(* IEC 61131-3 sources: ST_DesignPattern/Creational, 7 files *)

(* ---- abstract_factory_pattern.st ---- *)
{attribute 'qualified_only'}
{attribute 'strict'}
TYPE E_Color:
(
	init := 0,
	Black ,
	Red,
	Yellow,
	end
);
END_TYPE

{attribute 'qualified_only'}
{attribute 'strict'}
TYPE E_Shape:
(
	init := 0,
	Circle,
	Rectangle,
	Sqaure,
	Star,
	Triangle,
	end,
	Custom
);
END_TYPE

{attribute 'qualified_only'}
{attribute 'strict'}
TYPE E_Factory:
(
	init := 0,
	Shape,
	Color,
	end
);
END_TYPE

INTERFACE I_Color
    METHOD M_Fill: BOOL
    END_METHOD
END_INTERFACE

INTERFACE I_Shape
    METHOD M_Draw: BOOL
    END_METHOD
END_INTERFACE

FUNCTION_BLOCK FB_Black IMPLEMENTS I_Color
    METHOD M_Fill: BOOL
        ADSLOGSTR(ADSLOG_MSGTYPE_HINT, 'Paint Black', '');
        M_Fill := TRUE;
    END_METHOD
END_FUNCTION_BLOCK

FUNCTION_BLOCK FB_Red IMPLEMENTS I_Color
    METHOD M_Fill: BOOL
        ADSLOGSTR(ADSLOG_MSGTYPE_HINT, 'Paint Red', '');
        M_Fill := TRUE;
    END_METHOD
END_FUNCTION_BLOCK

FUNCTION_BLOCK FB_Yellow IMPLEMENTS I_Color
    METHOD M_Fill: BOOL
        ADSLOGSTR(ADSLOG_MSGTYPE_HINT, 'Paint Yellow', '');
        M_Fill := TRUE;
    END_METHOD
END_FUNCTION_BLOCK

FUNCTION_BLOCK FB_Circle IMPLEMENTS I_Shape
    METHOD M_Draw: BOOL
        ADSLOGSTR(ADSLOG_MSGTYPE_HINT, 'Draw circle', '');
        M_Draw := TRUE;
    END_METHOD
END_FUNCTION_BLOCK

FUNCTION_BLOCK FB_Rectangle IMPLEMENTS I_Shape
    METHOD M_Draw: BOOL
            ADSLOGSTR(ADSLOG_MSGTYPE_HINT, 'Draw rectangle', '');
            M_Draw := TRUE;
    END_METHOD
END_FUNCTION_BLOCK

FUNCTION_BLOCK FB_Sqaure IMPLEMENTS I_Shape
    METHOD M_Draw: BOOL
        ADSLOGSTR(ADSLOG_MSGTYPE_HINT, 'Draw square', '');
        M_Draw := TRUE;
    END_METHOD
END_FUNCTION_BLOCK

FUNCTION_BLOCK FB_Star IMPLEMENTS I_Shape
    METHOD M_Draw: BOOL
        ADSLOGSTR(ADSLOG_MSGTYPE_HINT, 'Draw star', '');
        M_Draw := TRUE;
    END_METHOD
END_FUNCTION_BLOCK

FUNCTION_BLOCK FB_Triangle IMPLEMENTS I_Shape
    METHOD M_Draw: BOOL
        ADSLOGSTR(ADSLOG_MSGTYPE_HINT, 'Draw triangle', '');
        M_Draw := TRUE;
    END_METHOD
END_FUNCTION_BLOCK

FUNCTION_BLOCK ABSTRACT FB_AbstractFactory
    METHOD M_GetColorObject: I_Color
    VAR_INPUT
        eColor: E_Color;
    END_VAR
    END_METHOD

    METHOD M_GetShapeObject: I_Shape
    VAR_INPUT
        eShape: E_Shape;
    END_VAR
    END_METHOD

    METHOD ABSTRACT M_ReleaseMemory: BOOL
    END_METHOD
END_FUNCTION_BLOCK

{attribute 'hide_all_locals'}
{attribute 'enable_dynamic_creation'}
FUNCTION_BLOCK FB_ColorCreator EXTENDS FB_AbstractFactory
    VAR
        pBlack: POINTER TO FB_Black;
        pRed: POINTER TO FB_Red;
        pCircle: POINTER TO FB_Circle;
        iColor: I_Color;
    END_VAR
    METHOD M_GetColorObject: I_Color
    VAR_INPUT
        eColor: E_Color;
    END_VAR
        CASE eColor OF:
            Black:

                // Dynamic instantiation
                pBlack := __NEW(FB_Black);
                iColor := pBlack^;

                // Return the object
                IF iColor <> 0 THEN
                    M_GetColorObject := iColor;
                END_IF

                eColor := E_Color.init;

            Red:

                // Dynamic instantiation
                pRed := __NEW(FB_Red);
                iColor := pRed^;

                // Return the object
                IF iColor <> 0 THEN
                    M_GetColorObject := iColor;
                END_IF

                eColor := E_Color.init;

            Yellow:

                // Dynamic instantiation
                pYellow := __NEW(FB_Yellow);
                iColor := pYellow^;

                // Return the object
                IF iColor <> 0 THEN
                    M_GetColorObject := iColor;
                END_IF

                eColor := E_Color.init;
        END_CASE
    END_METHOD

    METHOD M_ReleaseMemory
        // Release the memory
        IF (pBlack <> 0) THEN
            __DELETE(pBlack);
            pBlack := 0;
        END_IF

        // Release the memory
        IF (pRed <> 0) THEN
            __DELETE(pRed);
            pRed := 0;
        END_IF

        // Release the memory
        IF (pYellow <> 0) THEN
            __DELETE(pYellow);
            pYellow := 0;
        END_IF
    END_METHOD

    METHOD FB_exit
        M_ReleaseMemory();
    END_METHOD
END_FUNCTION_BLOCK

{attribute 'hide_all_locals'}
{attribute 'enable_dynamic_creation'}
FUNCTION_BLOCK FB_ShapeCreator EXTENDS FB_AbstractFactory
VAR
      pCircle: POINTER TO FB_Circle;
      pRectangle: POINTER TO FB_Rectangle;
      pSquare: POINTER TO FB_Square;
      pStar: POINTER TO FB_Star;
      pTriangle: POINTER TO FB_Triangle;
      iShape: I_Shape;
END_VAR

    METHOD M_GetShapeObject: I_shape
    VAR_INPUT
        eShape: E_Shape;
    END_VAR
        CASE eShape OF
            E_Shape.Circle:

                // Dynamic instantiation
                pCircle := __NEW(FB_Circle);
                iShape := pCircle^;

                // Return the object
                IF iShape <> 0 THEN
                    M_GetShapeObject := iShape;
                END_IF

                // Release the memory
                IF (pCircle <> 0) THEN
                    __DELETE(pCircle);
                    pCircle := 0;
                END_IF

                eShape := E_Shape.init;

            E_Shape.Rectangle:
                pRectangle := __NEW(FB_Rectangle);
                iShape := pRectangle^;

                // Return the object
                IF iShape <> 0 THEN
                    M_GetShapeObject := iShape;
                END_IF

                IF (pRectangle <> 0) THEN
                    __DELETE(pRectangle);
                    pRectangle := 0;
                END_IF

                eShape := E_Shape.init;

            E_Shape.Sqaure:
                pSquare := __NEW(FB_Square);
                iShape := pSquare^;

                // Return the object
                IF iShape <> 0 THEN
                    M_GetShapeObject := iShape;
                END_IF

                IF (pSquare <> 0) THEN
                    __DELETE(pSquare);
                    pSquare := 0;
                END_IF

                eShape := E_Shape.init;

            E_Shape.Star:
                pStar := __NEW(FB_Star);
                iShape := pStar^;

                // Return the object
                IF iShape <> 0 THEN
                    M_GetShapeObject := iShape;
                END_IF

                IF (pStar <> 0) THEN
                    __DELETE(pStar);
                    pStar := 0;
                END_IF

                eShape := E_Shape.init;

            E_Shape.Triangle:
                pTriangle := __NEW(FB_Triangle);
                iShape := pTriangle^;

                // Return the object
                IF iShape <> 0 THEN
                    M_GetShapeObject := iShape;
                END_IF

                IF (pTriangle <> 0) THEN
                    __DELETE(pTriangle);
                    pTriangle := 0;
                END_IF

                eShape := E_Shape.init;
        END_CASE
    END_METHOD

    METHOD M_ReleaseMemory: BOOL
    VAR_INPUT
    END_VAR
        IF (pCircle <> 0) THEN
            __DELETE(pCircle);
            pCircle := 0;
        END_IF

        IF (pRectangle <> 0) THEN
            __DELETE(pRectangle);
            pRectangle := 0;
        END_IF

        IF (pSquare <> 0) THEN
            __DELETE(pSquare);
            pSquare := 0;
        END_IF

        IF (pStar <> 0) THEN
            __DELETE(pStar);
            pStar := 0;
        END_IF

        IF (pTriangle <> 0) THEN
            __DELETE(pTriangle);
            pTriangle := 0;
        END_IF
    END_METHOD

    METHOD FB_exit: BOOL
    VAR_INPUT
        bInCopyCode: BOOL; // if TRUE, the exit method is called for exiting an instance that is copied afterwards (online change).
    END_VAR
        M_ReleaseMemory();
    END_METHOD
END_FUNCTION_BLOCK

FUNCTION_BLOCK FB_ShapeCreatorEX EXTENDS FB_ShapeCreator
VAR
	pCustomShape: POINTER TO FB_CustomShape;
END_VAR
    METHOD M_GetShapeObject: I_shape
        IF eShape = E_Shape.Custom THEN

            // Dynamic instantiation
            pCustomShape := __NEW(FB_CustomShape);
            iShape := pCustomShape^;

            // Return the object
            IF iShape <> 0 THEN
                M_GetShapeObject := iShape;
            END_IF

            // Release the memory
            IF (pCustomShape <> 0) THEN
                __DELETE(pCustomShape);
                pCustomShape := 0;
            END_IF

            eShape := E_Shape.init;
        ELSE
            M_GetShapeObject := SUPER^.M_GetShapeObject(eShape);
        END_IF
    END_METHOD
END_FUNCTION_BLOCK

FUNCTION_BLOCK FB_FactoryProducer
VAR
    pColorFactory: POINTER TO FB_ColorCreator;
    pShapeFactory: POINTER TO FB_ShapeCreator;
END_VAR
    METHOD M_GetFactory: REFERENCE TO FB_AbstractFactory
    VAR_INPUT
        eFactory: E_Factory;
    END_VAR
        CASE eFactory OF
            E_Factory.Color:

                pColorFactory := __NEW(FB_ColorCreator);
                IF pColorFactory <> 0 THEN
                    M_GetFactory REF= (pColorFactoy^);
                END_IF

                eFactory := E_Factory.init;

            E_Factory.Shape:

                pShapeFactory := __NEW(FB_ShapeCreator);
                IF pShapeFactory <> 0 THEN
                    M_GetFactory REF = (pShapeFactory^);
                END_IF

                eFactory := E_Factory.init;
        END_CASE
    END_METHOD

    METHOD M_ReleaseMemory: BOOL
        IF pColorFactoy <> 0 THEN
            __DELETE(pColorFactoy);
            pColorFactoy := 0;
        END_IF

        IF pShapeFactory <> 0 THEN
            __DELETE(pShapeFactory);
            pShapeFactory := 0;
        END_IF
    END_METHOD

    METHOD FB_exit: BOOL
    VAR_INPUT
        bInCopyCode: BOOL; // if TRUE, the exit method is called for exiting an instance that is copied afterwards (online change).
    END_VAR
        M_ReleaseMemory();
    END_METHOD
END_FUNCTION_BLOCK

PROGRAM MAIN
VAR
    fbFactoryProducer: FB_FactoryProducer;
    fbFactory: REFERENCE TO FB_AbstractFactory;

    iShape: I_Shape;
    iColor: I_Color;

    eShape: E_Shape := E_Shape.Star;
    eColor: E_Color := E_Color.Red;

    bStart1: BOOL;
    bStart2: BOOL;
END_VAR

IF bStart1 THEN
    // Draw
    fbFactory REF = fbFactoryProducer.M_GetFactory(eFactory := E_Factory.Shape);

    IF __ISVALIDREF(fbFactory) THEN
        iShape := fbFactory.M_GetShapeObject(eShape := eShape);
    END_IF

    IF iShape <> 0 THEN
		iShape.M_Draw();
	END_IF

    // Fill
    fbFactory REF = fbFactoryProducer.M_GetFactory(eFactory := E_Factory.Color);

    IF __ISVALIDREF(fbFactory) THEN
        iColor := fbFactory.M_GetColorObject(eColor := eColor);
    END_IF

    IF iColor <> 0 THEN
		iColor.M_Fill();
	END_IF

    // Release Memory
    fbFactoryProducer.M_ReleaseMemory();

    bStart1 := FALSE;
END_IF
// Alternatively, you can chain the methods and get the same result:
IF bStart2 THEN
	fbFactoryProducer.M_GetFactory(eFactory := E_Factory.Shape).M_GetShapeObject(eShape := eShape).M_Draw();
	fbFactoryProducer.M_GetFactory(eFactory := E_Factory.Color).M_GetColorObject(eColor := eColor).M_Fill();

	// Release Memory
	fbFactoryProducer.M_ReleaseMemory();
	bStart2 := FALSE;
END_IF
END_PROGRAM

(* ---- builder_patter_example1.st ---- *)
///The class Product is just a plain bluprint of the components of the object to be built.
///The final Product may ot may not contain the all the Parts listed on the Product declaration
/// rather only the parts in the specifications sent by the client.
{attribute 'enable_dynamic_creation' := ''}
FUNCTION_BLOCK Product
VAR_INPUT
	///List of possible parts to be build in a final Product object
	mainPart: STRING;
	part1: STRING;
	part2: STRING;
	part3: STRING;
END_VAR
    ///Method to be used in the visualization element for an easier String handling
    METHOD toString : STRING
    VAR
        ///Local variable to join together and store the pieces of String
        tempString: STRING;
    END_VAR
        //tempString joins together "Main Part" and "Part 1" of the Product object
        tempString := CONCAT(THIS^.mainPart , THIS^.part1);
        //tempString joins together its current value and "Part 2" of the Product object
        tempString := CONCAT(tempString , THIS^.part2);
        //tempString joins together its current value and "Part 3" of the Product object
        tempString := CONCAT(tempString , THIS^.part3);
        //The final result is sent as the output of this method
        toString := tempString;
    END_METHOD
END_FUNCTION_BLOCK

///Builder interface to declare all needed parts to be built
INTERFACE ITF_Builder
    ///Illustrative method of the pattern to set the main part
    METHOD Set_Main_Part
    VAR_INPUT
        ///Illustrative value (object because it is a TRING) to be set as a product part
        mainPart: STRING;
    END_VAR

    ///Illustrative method of the pattern to set the part1
    METHOD Set_Part1
    VAR_INPUT
        ///Illustrative value (object because it is a TRING) to be set as a product part
        part1: STRING;
    END_VAR

    ///Illustrative method of the pattern to set the part2
    METHOD Set_Part2
    VAR_INPUT
        ///Illustrative value (object because it is a TRING) to be set as a product part
        part2: STRING;
    END_VAR

    ///Illustrative method of the pattern to set the part3
    METHOD Set_Part3
    VAR_INPUT
        ///Illustrative value (object because it is a TRING) to be set as a product part
        part3: STRING;
    END_VAR
END_INTERFACE

///This is the concrete builder class, reponsible for building the final product object
FUNCTION_BLOCK ConcreteBuilder IMPLEMENTS ITF_Builder
VAR
	///Holds an internal reference to how the final product shoud be so the builder class can build it on the fly /// Contiene una referencia interna sobre cómo debe ser el producto final para que la clase constructora pueda construirlo sobre la marcha.
	/// without any help from other classes exepting the Director class that is going to be passing the special /// sin ninguna ayuda de otras clases excepto la clase Director que va a pasar el especial
	///specifications to the builder.///especificaciones para el constructor.
	localProduct: Product;
	///Stores the specifications, sent by the client, of the final product to be built.
	///Almacena las especificaciones, enviadas por el cliente, del producto final a construir.
	specifications: ARRAY[1..4] OF STRING;
END_VAR

METHOD fb_init
VAR_INPUT
	/// TRUE: the Retain-variables are initialized (reset warm / reset cold)
	bInitRetains: BOOL;
	/// TRUE  the instance will be copied to the copy-code afterward (online change)
	bInCopyCode: BOOL;
	///The constructor receives the specifications for this ConcreteBuilder instance
	///Just in case the concrete builder could change the specifications in the future, otherwise
	/// this specifications should be constant.
	specs: ARRAY[1..4] OF STRING;
END_VAR

    //Stores the specifications on its own specifications field.
    THIS^.specifications := specs;

END_METHOD

///Illustrative method of the pattern to get the main part
METHOD Get_Main_Part : STRING
    //Returns the object stored in the built product THIS^.localProduct.mainPart
    Get_Main_Part := THIS^.localProduct.mainPart;
END_METHOD

///Illustrative method of the pattern
METHOD Get_Result : Product
    //The concrete builder, after it builts the final object of class product, returns the
    // final product object
    Get_Result := THIS^.localProduct;
END_METHOD

///Illustrative method of the pattern to set the part1
METHOD Set_Part1
VAR_INPUT
	///Illustrative value (object because it is a TRING) to be set as a product part
	part1: STRING;
END_VAR
    //Sets the passed value to its corresponding field.
    //We can say that the the final product is in process of being built.
    //So this is a step into building the final product done by the builder.
    THIS^.localProduct.part1 := part1;
END_METHOD

END_FUNCTION_BLOCK

///The director class is responsible to delegate the construction of the final product object
/// to a concrete builder object.
{attribute 'enable_dynamic_creation' := ''}
FUNCTION_BLOCK Director
VAR_INPUT
	///Reference to the builder that is going to be building the final product object.
	///Referencia al constructor que construirá el objeto del producto final.
	{attribute 'old_input_assignments' := ''}
	inputConcreteBuilder: ConcreteBuilder(specs := inputConcreteBuilder.specifications);
END_VAR
VAR
	///Holds a reference to the concrete builder object to send the specifications of the final product to it.
	/// Contiene una referencia al objeto constructor concreto para enviarle las especificaciones del producto final
	{attribute 'old_input_assignments' := ''}
	concreteBuilder: ConcreteBuilder(specs := THIS^.concreteBuilder.specifications);
END_VAR
    //Stores the reference to which builder will be building the final product object in its own field THIS^.concreteBuilder
    //Almacena la referencia a qué constructor construirá el objeto del producto final en su propio campo THIS^.concreteBuilder
    THIS^.concreteBuilder := inputConcreteBuilder;

///This constructor is called at instanciation it is necessary to instanciate the Director instance.
///The specifications of the concreteBuilder instance stored in the Director instance should be set first by the client
/// otherwise a Data Recursion error is caused
METHOD fb_init
VAR_INPUT
	/// TRUE: the Retain-variables are initialized (reset warm / reset cold)
	bInitRetains: BOOL;
	/// TRUE  the instance will be copied to the copy-code afterward (online change)
	bInCopyCode: BOOL;
	///Reference a concreteBuilder instance to instanciate the Director.
	{attribute 'old_input_assignments' := ''}
	inputConcreteBuilder: ConcreteBuilder(specs := defaultArray);
END_VAR
VAR
	///Variable to isntanciate the concreteBuilder instance on the input section. It does not affect the Directors instanciation.
	defaultArray: ARRAY[1..4] OF STRING := ['Default', 'Default', 'Default', 'Default'];
END_VAR
    //Creates the concreteBuilder instance that will be building the final product object in its own field THIS^.concreteBuilder
    //This instance is empty because we can not use Data Recursion with the inputConcreteInstance instanciation.
    //So this concreteBuilder instance should be changed by the client before a Construct() request is called on the Director for the first time only.
    THIS^.concreteBuilder := inputConcreteBuilder;
END_METHOD

///This method is going to be called by the client when a new Product object must be built
METHOD Construct : Product
    //The Director tells its concreteBuilder instance to build the final product step by step passing the specifications stored in the
    // concreteBuilder array THIS^.specifications[1..4]

    //Step 1 "Main Part"
    THIS^.concreteBuilder.Set_Main_Part(THIS^.concreteBuilder.specifications[1]);
    //Step 2 "Part 1"
    THIS^.concreteBuilder.Set_Part1(THIS^.concreteBuilder.specifications[2]);
    //Step 3 "Part 2"
    THIS^.concreteBuilder.Set_Part2(THIS^.concreteBuilder.specifications[3]);
    //Step 4 "Part 3"
    THIS^.concreteBuilder.Set_Part3(THIS^.concreteBuilder.specifications[4]);

    //Finally the concreteBuilder instance in the Director object delivers the final result as a Product object
    //Finalmente, la instancia de concreteBuilder en el objeto Director entrega el resultado final como un objeto Producto
    Construct := THIS^.concreteBuilder.Get_Result();
END_METHOD
END_FUNCTION_BLOCK

(* ---- factory_method_pattern.st ---- *)
INTERFACE ITF_Cyclic EXTENDS __SYSTEM.IQueryInterface
    METHOD Cycle() : BOOL;
END_INTERFACE

{attribute 'enable_dynamic_creation'}
FUNCTION_BLOCK BasicObject IMPLEMENTS ITF_Cyclic
    METHOD Cycle : BOOL
END_FUNCTION_BLOCK

INTERFACE ITF_Mover
    PROPERTY VELOCITY : LREAL GET SET
END_INTERFACE

INTERFACE ITF_Station
    PROPERTY Position : LREAL GET SET
END_INTERFACE

INTERFACE ITF_Track
    PROPERTY Length : LREAL GET SET
END_INTERFACE

{attribute 'enable_dynamic_creation'}
FUNCTION_BLOCK Mover IMPLEMENTS ITF_Cyclic, ITF_Mover
VAR
	myMaxVelo : LREAL;
END_VAR
    {warning 'add method implementation '}
    METHOD Cycle : BOOL
    END_METHOD

    PROPERTY Velocity : LREAL GET
        Velocity := myMaxVelo;
    END_PROPERTY

    PROPERTY Velocity : LREAL SET
        myMaxVelo := Velocity;
    END_PROPERTY
END_FUNCTION_BLOCK

{attribute 'enable_dynamic_creation'}
FUNCTION_BLOCK Station IMPLEMENTS ITF_Cyclic, ITF_Station
VAR
	MyTrackPosition : LREAL;
END_VAR
    {warning 'add method implementation '}
    METHOD Cycle : BOOL
    END_METHOD

    PROPERTY Position : LREAL GET
        Position := MyTrackPosition;
    END_PROPERTY

    PROPERTY Position : LREAL SET
        MyTrackPosition := Position;
    END_PROPERTY
END_FUNCTION_BLOCK

{attribute 'enable_dynamic_creation'}
FUNCTION_BLOCK Track IMPLEMENTS ITF_Cyclic, ITF_Track
VAR
	MyTrackLength : LREAL;
END_VAR
    {warning 'add method implementation '}
    METHOD Cycle : BOOL
    END_METHOD

    PROPERTY Length : LREAL GET
        Length := MyTrackLength;
    END_PROPERTY

    PROPERTY Length : LREAL SET
        MyTrackLength := Length;
    END_PROPERTY
END_FUNCTION_BLOCK

INTERFACE ITF_Factory
    METHOD Create : ITF_Cyclic
END_INTERFACE

FUNCTION_BLOCK Factory IMPLEMENTS ITF_Factory
VAR
	ObjPtr : POINTER TO BasicObject;
END_VAR
    METHOD Create : ITF_Cyclic
        ObjPtr := __NEW(BasicObject);
        Create := ObjPtr^;
    END_METHOD
END_FUNCTION_BLOCK

FUNCTION_BLOCK MoverFactory EXTENDS Factory
VAR
	ptrMover : POINTER TO Mover;
	itfMover : ITF_Mover;
END_VAR
    METHOD Create : ITF_Cyclic
        PtrMover := __NEW(Mover);
        Create := ptrMover^;
        IF __QUERYINTERFACE(Create,itfMover) THEN
            itfMover.Velocity := 4000.0;
        END_IF
    END_METHOD
END_FUNCTION_BLOCK

FUNCTION_BLOCK StationFactory EXTENDS Factory
VAR
	prtStation : POINTER TO Station;
	itfStation : ITF_Station;
END_VAR
    METHOD Create : ITF_Cyclic
        prtStation := __NEW(Station);
        Create := prtStation^;
        IF __QUERYINTERFACE(Create,itfStation) THEN
            itfStation.Position := 1250.0;
        END_IF
    END_METHOD
END_FUNCTION_BLOCK

FUNCTION_BLOCK TrackFactory EXTENDS Factory
VAR
	ptrTrack : POINTER TO Track;
	itfTrack : ITF_Track;
END_VAR
    METHOD Create : ITF_Cyclic
        ptrTrack := __NEW(Track);
        Create := ptrTrack^;
        IF __QUERYINTERFACE(Create,itfTrack) THEN
            itfTrack.Length := 2500.0;
        END_IF
    END_METHOD
END_FUNCTION_BLOCK

PROGRAM MAIN
VAR
	State: INT;
	XtsMoverFactory : MoverFactory;
	XtsStationFactory : StationFactory;
	XtsTrackFactory : TrackFactory;
	iFactory : ITF_Factory := XtsMoverFactory;
	XtsElements : ARRAY[0..8] OF ITF_Cyclic;

	iMover : ITF_Mover;
	MaxVelo : LREAL;
	xTest: BOOL;
END_VAR
    CASE State OF
	0:
		IF Initialise() THEN
			State := 1;
		END_IF
    END_CASE

    IF xTest THEN
        xTest := FALSE;
        IF __QUERYINTERFACE(XtsElements[1],iMover) THEN
            MaxVelo := iMover.Velocity;
        END_IF
    END_IF

    METHOD Initialise : BOOL
    VAR
        i: INT;
    END_VAR
        FOR i := 0 TO 2 DO
            XtsElements[i] := iFactory.Create();
        END_FOR
        iFactory := XtsStationFactory;
        FOR i := 3 TO 5 DO
            XtsElements[i] := iFactory.Create();
        END_FOR
        iFactory := XtsTrackFactory;
        FOR i := 6 TO 8 DO
            XtsElements[i] := iFactory.Create();
        END_FOR
        Initialise := TRUE;
    END_METHOD
END_PROGRAM

(* ---- factory_method_pattern_example2.st ---- *)
{attribute 'qualified_only'}
{attribute 'strict'}
TYPE E_Shape :
(
	init := 0,
	Circle,
	Rectangle,
	Sqaure,
	Star,
	Triangle,
	end,
	Custom
);
END_TYPE

INTERFACE I_Shape
    METHOD M_Draw : BOOL
    END_METHOD
END_INTERFACE

{attribute 'enable_dynamic_creation'}
FUNCTION_BLOCK FB_Circle IMPLEMENTS I_Shape
    METHOD M_Draw : BOOL
        ADSLOGSTR(ADSLOG_MSGTYPE_HINT, 'Draw circle', '');
        M_Draw := TRUE;
    END_METHOD
END_FUNCTION_BLOCK

{attribute 'hide_all_locals'}
FUNCTION_BLOCK FB_ShapeCreator
VAR_INPUT
	eShape : E_Shape;
END_VAR
VAR
      pCircle    : POINTER TO FB_Circle;
      pRectangle : POINTER TO FB_Rectangle;
      pSquare    : POINTER TO FB_Square;
      pStar      : POINTER TO FB_Star;
      pTriangle  : POINTER TO FB_Triangle;
      iShape 	 : I_Shape;
END_VAR
    METHOD M_GetShapeObject : I_shape
        CASE eShape OF
            E_Shape.Circle:

                //Dynamic instantiation
                pCircle := __NEW(FB_Circle);
                iShape := pCircle^;

                //Return the object
                IF iShape <> 0 THEN
                    M_GetShapeObject := iShape;
                END_IF

                //Release the memory
                IF (pCircle <> 0) THEN
                    __DELETE(pCircle);
                    pCircle := 0;
                END_IF

                eShape := E_Shape.init;

            E_Shape.Rectangle:
                pRectangle := __NEW(FB_Rectangle);
                iShape := pRectangle^;

                //Return the object
                IF iShape <> 0 THEN
                    M_GetShapeObject := iShape;
                END_IF

                IF (pRectangle <> 0) THEN
                    __DELETE(pRectangle);
                    pRectangle := 0;
                END_IF

                eShape := E_Shape.init;
            // TODO: others
        END_CASE
    END_METHOD

    METHOD M_ReleaseMemory : BOOL
    END_METHOD
    METHOD FB_exit : BOOL
    END_METHOD
END_FUNCTION_BLOCK

PROGRAM MAIN
VAR
	//fbShapeCreator : FB_ShapeCreator;
	fbShapeCreator : FB_ShapeCreatorEX;
	eShape : E_Shape := E_Shape.init;

	iShape : I_Shape;
END_VAR

    fbShapeCreator(eShape:= eShape);
    CASE eShape OF
        E_Shape.Circle:
            iShape := fbShapeCreator.M_GetShapeObject();
            IF iShape <> 0 THEN
                iShape.M_Draw();
            END_IF

            eShape := E_Shape.Rectangle;

        E_Shape.Rectangle:
            iShape := fbShapeCreator.M_GetShapeObject();
            IF iShape <> 0 THEN
                iShape.M_Draw();
            END_IF

            eShape := E_Shape.Sqaure;
        // TODO: Complete rest
    END_CASE
END_PROGRAM

(* ---- observer_pattern.st ---- *)
{attribute 'qualified_only'}
{attribute 'strict'}
TYPE E_OperationType :
(
    UNKNOWN := 0,
    VALVE,
    MFC_SET,
    MFC_WAIT,
    PRESSURE_WAIT,
    TIMER_WAIT,
    LOOP
);
END_TYPE

{attribute 'strict'}
TYPE ST_OperationData :
STRUCT
    eOperation : E_OperationType;
    eValve : E_Valve; // Assuming E_Valve is defined elsewhere
    bOpen : BOOL;
    rSetPoint : REAL;
    tTimeout : TIME;
    tStabilizationTime : TIME;
    rFlowTolerance : REAL;
    bResetLoop : BOOL;
    nCurrentCycle : DINT;
    nMaxCycles : DINT;
    eLoopNextState : E_PurgeState; // Assuming E_PurgeState is defined elsewhere
    eLoopStartState : E_PurgeState;
    eNextState : E_PurgeState;
    eErrorState : E_ErrorState; // Assuming E_ErrorState is defined elsewhere
    eCategory : E_ErrorCategory; // Assuming E_ErrorCategory is defined elsewhere
    eErrorCode : E_ErrorCodes; // Assuming E_ErrorCodes is defined elsewhere
    sDescription : STRING;
    sCurrentValue : STRING;
    sExpectedValue : STRING;
    sUnit : STRING;
    bAbove: BOOL;
    rTolerance: REAL;
END_STRUCT
END_TYPE

INTERFACE I_Operation
METHOD Execute : BOOL
VAR_INPUT
    fbErrorHandler : REFERENCE TO FB_ErrorHandler;
END_VAR
    METHOD Reset : BOOL
VAR_INPUT
END_VAR
END_INTERFACE

FUNCTION_BLOCK ABSTRACT FB_BaseOperation IMPLEMENTS I_Operation
VAR
    _bDone : BOOL;
    _bError : BOOL;
    _eNextState : E_PurgeState;
END_VAR

METHOD ABSTRACT Execute : BOOL
VAR_INPUT
    fbErrorHandler : REFERENCE TO FB_ErrorHandler;
END_VAR
END_METHOD

METHOD Reset : BOOL
VAR_INPUT
END_VAR
    _bDone := FALSE;
    _bError := FALSE;
    Reset := TRUE;
END_METHOD

FUNCTION_BLOCK FB_ValveOperation EXTENDS FB_BaseOperation
VAR
    _fbValveManager: REFERENCE TO FB_ValveManager;
    _eValve : E_Valve;
    _bOpen : BOOL;
END_VAR

METHOD SetParameters : BOOL
VAR_INPUT
    fbValveManager: REFERENCE TO FB_ValveManager;
    eValve : E_Valve;
    bOpen : BOOL;
END_VAR
    _fbValveManager REF= fbValveManager;
    _eValve := eValve;
    _bOpen := bOpen;
    SetParameters := TRUE;
END_METHOD

METHOD Execute: BOOL
VAR_INPUT
    fbErrorHandler : REFERENCE TO FB_ErrorHandler;
END_VAR
VAR
    stError: ST_Error;
    stValveStatus: ST_ValveStatus;
END_VAR
    // Reset state
    _bDone := FALSE;
    _bError := FALSE;

    // Perform valve operation
    IF _bOpen THEN
        _fbValveManager.OpenValve(_eValve);
    ELSE
        _fbValveManager.CloseValve(_eValve);
    END_IF

    // Check valve status
    stValveStatus := _fbValveManager.GetValveStatus(_eValve);
    IF stValveStatus.bError THEN
        stError := stValveStatus.stError;
        fbErrorHandler.UpdateError(stError);
        _bError := TRUE;
        RETURN FALSE;
    END_IF

    // Check if valve operation is complete
    _bDone := NOT stValveStatus.bBusy;

    Execute := _bDone AND NOT _bError;
END_METHOD

INTERFACE I_OperationDecorator IMPLEMENTS I_Operation
END_INTERFACE

FUNCTION_BLOCK FB_TimeoutDecorator IMPLEMENTS I_OperationDecorator
VAR
    _operation : I_Operation;
    _tTimeout : TIME;
    _fbTimerManager : FB_TimerManager;
    _stOperationData : ST_OperationData;
END_VAR

METHOD SetParameters : BOOL
VAR_INPUT
    operation : I_Operation;
    tTimeout : TIME;
    stOperationData : ST_OperationData;
END_VAR
    _operation := operation;
    _tTimeout := tTimeout;
    _stOperationData := stOperationData;
    SetParameters := TRUE;
END_METHOD

METHOD Execute : BOOL
VAR_INPUT
    fbErrorHandler : REFERENCE TO FB_ErrorHandler;
END_VAR
VAR
    bTimedOut : BOOL;
    stError : ST_Error;
END_VAR
    // Update timers
    _fbTimerManager.Update();

    // Start operation timer if not active
    IF NOT _fbTimerManager.StartOperationTimer(_tTimeout) THEN
        _fbTimerManager.StartOperationTimer(_tTimeout);
    END_IF

    // Check for operation timeout
    IF _fbTimerManager.IsOperationTimeout() THEN
        stError.eCategory := E_ErrorCategory.Timeout; // Assuming E_ErrorCategory is defined elsewhere
        stError.eErrorCode := E_ErrorCodes.OperationTimeout; // Assuming E_ErrorCodes is defined elsewhere
        stError.sComponent := 'FB_TimeoutDecorator';
        stError.sDescription := 'Operation timeout';
        fbErrorHandler.UpdateError(stError);
        RETURN FALSE;
    END_IF

    // Execute the decorated operation
    Execute := _operation.Execute(fbErrorHandler := fbErrorHandler);
END_METHOD

METHOD Reset : BOOL
VAR_INPUT
END_VAR
    _fbTimerManager.Reset();
    Reset := TRUE;
END_METHOD

FUNCTION_BLOCK FB_StabilizationDecorator IMPLEMENTS I_OperationDecorator
VAR
    _operation : I_Operation;
    _tStabilizationTime : TIME;
    _fbTimerManager : FB_TimerManager;
    _bConditionMet : BOOL;
    _stOperationData : ST_OperationData;
END_VAR

METHOD SetParameters : BOOL
VAR_INPUT
    operation : I_Operation;
    tStabilizationTime : TIME;
    bConditionMet : BOOL;
    stOperationData : ST_OperationData;
END_VAR
    _operation := operation;
    _tStabilizationTime := tStabilizationTime;
    _bConditionMet := bConditionMet;
    _stOperationData := stOperationData;
    SetParameters := TRUE;
END_METHOD

METHOD Execute : BOOL
VAR_INPUT
    fbErrorHandler : REFERENCE TO FB_ErrorHandler;
END_VAR
VAR
    bStabilizationComplete : BOOL;
END_VAR
    // Execute the decorated operation
    IF NOT _operation.Execute(fbErrorHandler := fbErrorHandler) THEN
        Execute := FALSE;
        RETURN FALSE;
    END_IF

    // Start stabilization timer if condition met
    _fbTimerManager.StartStabilizationTimer(_tStabilizationTime, _bConditionMet);

    // Check if operation is complete
    bStabilizationComplete := _fbTimerManager.IsStabilizationComplete();
    IF bStabilizationComplete THEN
        Execute := TRUE;
    ELSE
        Execute := FALSE;
    END_IF
END_METHOD

METHOD Reset : BOOL
VAR_INPUT
END_VAR
    _fbTimerManager.Reset();
    Reset := TRUE;
END_METHOD

FUNCTION_BLOCK FB_OperationFactory
VAR
    _fbValveManager: REFERENCE TO FB_ValveManager;
    _fbValveOperation: POINTER TO FB_ValveOperation;
    _fbTimeoutDecorator : POINTER TO FB_TimeoutDecorator;
    _fbStabilizationDecorator : POINTER TO FB_StabilizationDecorator;
    _iOperation : I_Operation;
    _iTimeoutDecorator : I_OperationDecorator;
    _iStabilizationDecorator : I_OperationDecorator;
END_VAR

METHOD SetValveManager : BOOL
VAR_INPUT
    fbValveManager: REFERENCE TO FB_ValveManager;
END_VAR
    _fbValveManager REF= fbValveManager;
    SetValveManager := TRUE;
END_METHOD

METHOD CreateValveOperation : I_Operation
VAR_INPUT
    stOperationData : ST_OperationData;
    bWithTimeout : BOOL;
    bWithStabilization : BOOL;
END_VAR
    // Create Valve Operation
    _fbValveOperation := __NEW(FB_ValveOperation);
    _iOperation := _fbValveOperation^;
    _fbValveOperation^.SetParameters(
        fbValveManager := _fbValveManager,
        eValve := stOperationData.eValve,
        bOpen := stOperationData.bOpen
    );

    CreateValveOperation := _iOperation;

    IF bWithTimeout THEN
        _fbTimeoutDecorator := __NEW(FB_TimeoutDecorator);
        _iTimeoutDecorator := _fbTimeoutDecorator^;
        _fbTimeoutDecorator^.SetParameters(
            operation := CreateValveOperation,
            tTimeout := stOperationData.tTimeout,
            stOperationData := stOperationData
        );
        CreateValveOperation := _iTimeoutDecorator;
    END_IF;

    IF bWithStabilization THEN
        _fbStabilizationDecorator := __NEW(FB_StabilizationDecorator);
        _iStabilizationDecorator := _fbStabilizationDecorator^;
        _fbStabilizationDecorator^.SetParameters(
            operation := CreateValveOperation,
            tStabilizationTime := stOperationData.tStabilizationTime,
            bConditionMet := TRUE, // Set your condition here
            stOperationData := stOperationData
        );
        CreateValveOperation := _iStabilizationDecorator;
    END_IF;
END_METHOD

METHOD DeleteValveOperation : BOOL
VAR_INPUT
    bWithTimeout : BOOL;
    bWithStabilization : BOOL;
END_VAR
    IF _fbValveOperation <> 0 THEN
        __DELETE(_fbValveOperation);
        _fbValveOperation := 0;
    END_IF

    IF bWithTimeout AND _fbTimeoutDecorator <> 0 THEN
        __DELETE(_fbTimeoutDecorator);
        _fbTimeoutDecorator := 0;
    END_IF

    IF bWithStabilization AND _fbStabilizationDecorator <> 0 THEN
        __DELETE(_fbStabilizationDecorator);
        _fbStabilizationDecorator := 0;
    END_IF

    DeleteValveOperation := TRUE;
END_METHOD

INTERFACE I_OperationSequence
    METHOD AddOperation
    VAR_INPUT
        operation : I_Operation;
    END_VAR
    END_METHOD

    METHOD ExecuteAll : BOOL
    VAR_INPUT
         fbErrorHandler : REFERENCE TO FB_ErrorHandler;
    END_VAR
    END_METHOD

    METHOD ResetAll : BOOL
    END_METHOD
END_INTERFACE

FUNCTION_BLOCK FB_OperationSequence IMPLEMENTS I_OperationSequence
VAR
    _operations : ARRAY [1..10] OF I_Operation; // Assuming a max of 10 operations
    _operationCount : INT;
END_VAR

METHOD AddOperation
VAR_INPUT
    operation : I_Operation;
END_VAR
    _operationCount := _operationCount + 1;
    _operations[_operationCount] := operation;
END_METHOD

METHOD ExecuteAll : BOOL
VAR_INPUT
     fbErrorHandler : REFERENCE TO FB_ErrorHandler;
END_VAR
VAR
    i : INT;
    bResult : BOOL := TRUE;
END_VAR
    FOR i := 1 TO _operationCount DO
        IF _operations[i] <> 0 THEN
            bResult := bResult AND _operations[i].Execute(fbErrorHandler := fbErrorHandler);
        END_IF
    END_FOR
    ExecuteAll := bResult;
END_METHOD

METHOD ResetAll : BOOL
VAR
    i : INT;
END_VAR
    FOR i := 1 TO _operationCount DO
        IF _operations[i] <> 0 THEN
            _operations[i].Reset();
        END_IF
    END_FOR
    _operationCount := 0;
END_METHOD

PROGRAM MAIN
VAR
    fbOperationFactory : FB_OperationFactory;
    fbValveManager : FB_ValveManager; // Assuming FB_ValveManager is defined elsewhere
    fbOperationSequence : FB_OperationSequence;
    stOperationData1 : ST_OperationData;
    stOperationData2 : ST_OperationData;
    stOperationData3 : ST_OperationData;
    iValveOperation1 : I_Operation;
    iValveOperation2 : I_Operation;
    iValveOperation3 : I_Operation;
    bExecute : BOOL;
    bWithTimeout : BOOL := TRUE;
    bWithStabilization : BOOL := TRUE;
    fbErrorHandler : FB_ErrorHandler;
END_VAR

    // Initialize OperationFactory with ValveManager
    fbOperationFactory.SetValveManager(fbValveManager := fbValveManager);

    // Initialize operation data for Valve1
    stOperationData1.eOperation := E_OperationType.VALVE;
    stOperationData1.eValve := E_Valve.Valve1; // Assuming E_Valve.Valve1 is defined elsewhere
    stOperationData1.bOpen := TRUE;
    stOperationData1.tTimeout := T#5s;
    stOperationData1.tStabilizationTime := T#2s;

    // Create valve operation with timeout and stabilization for Valve1
    iValveOperation1 := fbOperationFactory.CreateValveOperation(
        stOperationData := stOperationData1,
        bWithTimeout := bWithTimeout,
        bWithStabilization := bWithStabilization
    );

     // Initialize operation data for Valve2
    stOperationData2.eOperation := E_OperationType.VALVE;
    stOperationData2.eValve := E_Valve.Valve2; // Assuming E_Valve.Valve2 is defined elsewhere
    stOperationData2.bOpen := FALSE;
    stOperationData2.tTimeout := T#3s;
    stOperationData2.tStabilizationTime := T#1s;

    // Create valve operation with timeout and stabilization for Valve2
    iValveOperation2 := fbOperationFactory.CreateValveOperation(
        stOperationData := stOperationData2,
        bWithTimeout := bWithTimeout,
        bWithStabilization := bWithStabilization
    );

     // Initialize operation data for Valve3
    stOperationData3.eOperation := E_OperationType.VALVE;
    stOperationData3.eValve := E_Valve.Valve3; // Assuming E_Valve.Valve3 is defined elsewhere
    stOperationData3.bOpen := TRUE;
    stOperationData3.tTimeout := T#4s;
    stOperationData3.tStabilizationTime := T#2s;

    // Create valve operation with timeout and stabilization for Valve3
    iValveOperation3 := fbOperationFactory.CreateValveOperation(
        stOperationData := stOperationData3,
        bWithTimeout := bWithTimeout,
        bWithStabilization := bWithStabilization
    );

    // Add operations to sequence
    fbOperationSequence.AddOperation(iValveOperation1);
    fbOperationSequence.AddOperation(iValveOperation2);
     fbOperationSequence.AddOperation(iValveOperation3);

    // Execute the sequence
    IF bExecute THEN
        bExecute := FALSE;
        fbOperationSequence.ExecuteAll(fbErrorHandler := fbErrorHandler);
    END_IF

    // Clean up memory
    fbOperationFactory.DeleteValveOperation(bWithTimeout := bWithTimeout ,bWithStabilization := bWithStabilization);
END_PROGRAM

(* ---- simple_factory_pattern.st ---- *)
INTERFACE I_EtherCATDevice
    METHOD IsDeviceOK : BOOL
END_INTERFACE

{attribute 'enable_dynamic_creation'}
FUNCTION_BLOCK EtherCATDevice IMPLEMENTS I_EtherCATDevice
    METHOD IsDeviceOK : BOOL
        IsDeviceOK := true;
    END_METHOD
END_FUNCTION_BLOCK

FUNCTION_BLOCK EtherCATFactory
    METHOD PUBLIC CreateEtherCATDevice : I_EtherCATDevice
        VAR
            devicePtr: POINTER TO EtherCATDevice;
        END_VAR
        devicePtr := __NEW(EtherCATDevice);
        CreateEtherCATDevice := devicePtr^;
    END_METHOD
END_FUNCTION_BLOCK

PROGRAM MAIN
VAR
	EtherCATIOFactory : EtherCATFactory;
	GetEtherCATDevice: BOOL;
	myDevcie : I_EtherCATDevice;
	CheckMyDevice: BOOL;
	value: BOOL;
END_VAR
    IF GetEtherCATDevice THEN
        GetEtherCATDevice := FALSE;
        myDevcie := EtherCATIOFactory.CreateEtherCATDevice();
    END_IF

    IF CheckMyDevice THEN
        CheckMyDevice := false;
        value := myDevcie.IsDeviceOK();
    END_IF
END_PROGRAM

(* ---- strategy_pattern.st ---- *)
INTERFACE ITF_Writer
    METHOD WriteMessage : BOOL
    VAR_INPUT
        SomeString : STRING(80);
    END_VAR
    END_METHOD
END_INTERFACE

FUNCTION_BLOCK CSVWriter IMPLEMENTS ITF_Writer
    METHOD WriteMessage : BOOL
    VAR_INPUT
        SomeString	: STRING(80);
    END_VAR
        ADSLOGSTR(msgCtrlMask := ADSLOG_MSGTYPE_LOG, msgFmtStr := 'I wrote a CSV line with: %s',strArg := SomeString);
    END_METHOD
END_FUNCTION_BLOCK

FUNCTION_BLOCK JsonWriter IMPLEMENTS ITF_Writer
    METHOD WriteMessage : BOOL
    VAR_INPUT
        SomeString	: STRING(80);
    END_VAR
        ADSLOGSTR(msgCtrlMask := ADSLOG_MSGTYPE_LOG, msgFmtStr := 'I wrote a JSON line with: %s',strArg := SomeString);
    END_METHOD
END_FUNCTION_BLOCK

FUNCTION_BLOCK TextWriter IMPLEMENTS ITF_Writer
    METHOD WriteMessage : BOOL
    VAR_INPUT
        SomeString	: STRING(80);
    END_VAR
        ADSLOGSTR(msgCtrlMask := ADSLOG_MSGTYPE_LOG, msgFmtStr := 'I wrote a Text line with: %s',strArg := SomeString);
    END_METHOD
END_FUNCTION_BLOCK

FUNCTION_BLOCK SomeCyclicClass
VAR
	_myWriter : ITF_Writer;
END_VAR
    METHOD DoSomething : BOOL
        ///////Perform some operations////////
        IF _myWriter <> 0 THEN
            _myWriter.WriteMessage('I did a job :-)');
        END_IF
    END_METHOD
    PROPERTY MyWriter : ITF_Writer
        GET
            MyWriter := _myWriter;
        SET
            _myWriter := MyWriter;
    END_PROPERTY
END_FUNCTION_BLOCK
